(* IEC 61131-3 sources: mapp-robotics-getting-started/, 1 file *)

(* ---- Robotic.st ---- *)
VAR CONSTANT
   P1 : McPointType := (Pos:=(X:=0, Y:=0, Z:=-650));
   P2 : McPointType := (Pos:=(X:=-50, Y:=-20, Z:=-600));
   P0 : McPointType := (Pos:=(X:=0, Y:=0, Z:=-560));
END_VAR

PROGRAM _MAIN
 Feedrate(5000);   //move with reduced speed
 MoveJ(P1);        //move system to point P1
MoveJ(P2);        //move system to point P2

 WaitTime(3);        //wait for 3 seconds

 MoveJ(P0);        //move back to origin position
END_PROGRAM
